// TwinCAT 3 PLC project TcLogger
// Title: TcLogger
// Company: TcLogger
// ProjectVersion: 0.2.0
// ProgramVersion: 3.1.4022.7
// libraries:
//   Tc2_Standard, * (Beckhoff Automation GmbH)
//   Tc2_System, * (Beckhoff Automation GmbH)
//   Tc2_Utilities, * (Beckhoff Automation GmbH)
//   Tc3_Module, * (Beckhoff Automation GmbH)
//   TcExt, * (TcExt)
//   TcUnit, * (www.tcunit.org)
// project tree:
//   Event/ Event.TcPOU (not stored), EventLevel.TcDUT, EventMessage.TcDUT (not stored), EventRunner.TcPOU
//   GVL/ GVL.TcGVL, Properties.TcGVL
//   Logger/ ADSLogger.TcPOU, EventLogger.TcIO, FileLogger.TcPOU, MemoryLogger.TcPOU, run.TcPOU
//   / PlcTask.TcTTO
//   Tests/Event/ EventTestsystem.TcDUT (not stored), MultipleEventTestsystem.TcDUT, TestEvent.TcPOU
//   Tests/Logger/ ADSLoggerTestsystem.TcDUT, TestADSLogger.TcPOU, TestFileLogger.TcPOU
//   Tests/ TEST_MAIN.TcPOU
//   Utils/ F_FIFO_WRITE.TcPOU (not stored), remove_field_from_array.TcPOU (not stored)
// real-time tasks:
//   TASK PlcTask: cycle T#10ms, priority 20, ADS port 350

CONFIGURATION TcLogger
    RESOURCE PLC ON TwinCAT3
        TASK PlcTask(INTERVAL := T#10ms, PRIORITY := 20);
        PROGRAM TEST_MAIN WITH PlcTask : TEST_MAIN;
    END_RESOURCE
END_CONFIGURATION

// ---- Event/EventLevel.TcDUT
{attribute 'qualified_only'}
{attribute 'strict'}
TYPE EventLevel :
(
	INFO := 10,
  WARNING :=20,
  ERROR := 30
) BYTE := INFO;
END_TYPE

// ---- Tests/Event/MultipleEventTestsystem.TcDUT
TYPE MultipleEventTestsystem :
STRUCT
  runner: EventRunner;
  event1: Event := (runner:=runner);
  event2: Event := (runner:=runner);
  event3: Event := (runner:=runner);
END_STRUCT
END_TYPE

// ---- Tests/Logger/ADSLoggerTestsystem.TcDUT
TYPE ADSLoggerTestsystem :
STRUCT
  runner: EventRunner;
  event: Event := (runner:=runner);
  logger: ADSLogger := (disable_ads_output := TRUE);
END_STRUCT
END_TYPE

// ---- GVL/GVL.TcGVL
{attribute 'qualified_only'}
VAR_GLOBAL
  runner: EventRunner;
END_VAR

// ---- GVL/Properties.TcGVL
{attribute 'qualified_only'}
VAR_GLOBAL CONSTANT
  NUM_EVENTS: INT := 4;
  NUM_EVENT_HISTORY: INT := 10;
  NUM_CONCURRENT_ALARMS: INT := 10;
  NUM_LOGGER: INT := 5;
END_VAR

// ---- Logger/EventLogger.TcIO
INTERFACE EventLogger

PROPERTY PUBLIC level : EventLevel
GET
END_GET
SET
END_SET
END_PROPERTY

METHOD PUBLIC submit_event_message
VAR_INPUT
  ev: EventMessage;
END_VAR
END_METHOD

END_INTERFACE

// ---- Tests/TEST_MAIN.TcPOU
PROGRAM TEST_MAIN
VAR
  test_event: TestEvent;
  test_ads_logger: TestADSLogger;
  //test_file_logger: TestFileLogger;
END_VAR

TcUnit.RUN();

END_PROGRAM

// ---- Tests/Event/TestEvent.TcPOU
FUNCTION_BLOCK TestEvent EXTENDS TcUnit.FB_TestSuite
VAR_INPUT
END_VAR
VAR_OUTPUT
END_VAR
VAR
END_VAR

event_erstellen();
//file_logger_testen();
after_initialisation_alarm_is_not_raised();
after_raising_an_alarm_the_alarm_is_raised();
clear_alarm();
add_multiple_events();
raise_and_clear_multiple_alarms();

METHOD add_multiple_events
VAR_INST
  sut: MultipleEventTestsystem;
END_VAR
TEST('Add multiple events');

sut.event1.alarm();
sut.event2.warning();
sut.event3.alarm();
AssertTrue(sut.event1.alarm_raised, 'Event 1');
AssertFalse(sut.event2.alarm_raised, 'Event 2');
AssertTrue(sut.event3.alarm_raised, 'Event 3');

TEST_FINISHED();
END_METHOD

METHOD after_initialisation_alarm_is_not_raised
VAR_INPUT
END_VAR
VAR_INST
  sut: EventTestsystem;
END_VAR
TEST('Alarm is not raised after initialisation');

AssertFalse(sut.event.alarm_raised, '');

TEST_FINISHED();
END_METHOD

METHOD after_raising_an_alarm_the_alarm_is_raised
VAR_INPUT
END_VAR
VAR_INST
  sut: EventTestsystem;
END_VAR
TEST('After raising an alarm the alarm is raised');

sut.event.alarm();
AssertTrue(sut.event.alarm_raised, '');

TEST_FINISHED();
END_METHOD

METHOD clear_alarm
VAR_INPUT
END_VAR
VAR_INST
  sut: EventTestsystem;
END_VAR
TEST('Clear alarm');

sut.event.alarm();
sut.event.clear_alarm();
AssertFalse(sut.event.alarm_raised, '');

TEST_FINISHED();
END_METHOD

METHOD event_erstellen
VAR_INPUT
END_VAR
VAR_INST
  sut: EventTestsystem;
END_VAR
TEST('event_erstellen');

sut.event.message := 'Test';
AssertEquals_STRING('Test', sut.event.message, 'Event not properly created');

TEST_FINISHED();
END_METHOD

METHOD file_logger_testen
VAR_INPUT
END_VAR
VAR_INST
  sut: EventTestsystem;
  file_logger: FileLogger;
END_VAR
TEST('file_logger_testen');

file_logger.path := 'c:\';
sut.runner.add_logger(file_logger);
sut.event.message := 'Test';
sut.event.alarm();

//sut.runner.save_logger(execute:=TRUE);

//IF sut.runner.saving_logger_done() THEN
  TEST_FINISHED();
//END_IF
END_METHOD

METHOD raise_and_clear_multiple_alarms
VAR_INST
  sut: MultipleEventTestsystem;
END_VAR
TEST('Raise and clear multiple alarms');

sut.event1.alarm();
sut.event2.alarm();
sut.event3.alarm();
sut.event1.clear_alarm();
sut.event3.clear_alarm();
AssertFalse(sut.event1.alarm_raised, 'Event 1');
AssertTrue(sut.event2.alarm_raised, 'Event 2');
AssertFalse(sut.event3.alarm_raised, 'Event 3');

TEST_FINISHED();
END_METHOD

END_FUNCTION_BLOCK

// ---- Logger/FileLogger.TcPOU
FUNCTION_BLOCK FileLogger IMPLEMENTS EventLogger
VAR_INPUT
END_VAR
VAR_OUTPUT
  error_id: DWORD;
END_VAR
VAR
  _path: STRING(255);
  file: TcExt.FileMemory;
  localtime: FB_LocalSystemTime := (bEnable:=TRUE);
  _done: BOOL;
  _level: EventLevel;
END_VAR

PROPERTY done : BOOL
GET
done := _done;
END_GET
SET // PRIVATE
_done := done;
END_SET
END_PROPERTY

METHOD PRIVATE get_timestaped_path : STRING(255)
VAR
  datetime: STRING(255);
  char_at: INT;
END_VAR
datetime := SYSTEMTIME_TO_STRING(localtime.systemTime);

char_at := FIND(datetime, '.');
IF char_at <> 0 THEN
  datetime := DELETE(datetime, 4, char_at);
END_IF

REPEAT
  char_at := FIND(datetime, ':');
  IF char_at <> 0 THEN
    datetime := REPLACE(datetime, '_', 1, char_at);
  END_IF
UNTIL char_at = 0
END_REPEAT

get_timestaped_path := CONCAT(path, CONCAT('log_', CONCAT(datetime, '.log')));
END_METHOD

PROPERTY PUBLIC level : EventLevel
GET
level := _level;
END_GET
SET
_level := level;
END_SET
END_PROPERTY

PROPERTY path : STRING(255)
GET
path := _path;
END_GET
SET
_path := path;
END_SET
END_PROPERTY

METHOD save
VAR_INPUT
  execute: BOOL;
  data_ptr: PVOID;
  data_size: DWORD;
END_VAR
VAR_INST
  r_execute: R_TRIG;
END_VAR
localtime();
r_execute(CLK:=execute);

IF r_execute.Q THEN
  file.path := get_timestaped_path();
END_IF
file.write(
  start:=execute,
  data_ptr:=data_ptr,
  data_size:=data_size,
  done=>_done,
  error_id=>error_id);
END_METHOD

METHOD submit_event_message
VAR_INPUT
	ev: EventMessage;
END_VAR
END_METHOD

END_FUNCTION_BLOCK

// ---- Tests/Logger/TestADSLogger.TcPOU
FUNCTION_BLOCK TestADSLogger EXTENDS TcUnit.FB_TestSuite
VAR_INPUT
END_VAR
VAR_OUTPUT
END_VAR
VAR
END_VAR

submit_info();
submit_warning();
submit_error();
submit_alarm();

METHOD submit_alarm
VAR_INPUT
END_VAR
VAR_INST
  sut: ADSLoggerTestsystem;
END_VAR
TEST('Submit alarm');

sut.runner.add_logger(sut.logger);
sut.event.message := 'Alarm';
sut.event.alarm();

AssertEquals_DWORD(ADSLOG_MSGTYPE_ERROR, sut.logger.mask, '');
AssertEquals_STRING(' | Error: ', sut.logger.prefix, '');
AssertEquals_STRING(' | Error: Alarm', sut.logger.formatted_output, '');

TEST_FINISHED();
END_METHOD

METHOD submit_error
VAR_INPUT
END_VAR
VAR_INST
  sut: ADSLoggerTestsystem;
END_VAR
TEST('Submit error');

sut.runner.add_logger(sut.logger);
sut.event.message := 'Error';
sut.event.error();

AssertEquals_DWORD(ADSLOG_MSGTYPE_ERROR, sut.logger.mask, '');
AssertEquals_STRING(' | Error: ', sut.logger.prefix, '');
AssertEquals_STRING(' | Error: Error', sut.logger.formatted_output, '');

TEST_FINISHED();
END_METHOD

METHOD submit_info
VAR_INPUT
END_VAR
VAR_INST
  sut: ADSLoggerTestsystem;
END_VAR
TEST('Submit info');

sut.runner.add_logger(sut.logger);
sut.event.message := 'Info';
sut.event.info();

AssertEquals_DWORD(ADSLOG_MSGTYPE_HINT, sut.logger.mask, '');
AssertEquals_STRING(' | Info: ', sut.logger.prefix, '');
AssertEquals_STRING(' | Info: Info', sut.logger.formatted_output, '');

TEST_FINISHED();
END_METHOD

METHOD submit_warning
VAR_INPUT
END_VAR
VAR_INST
  sut: ADSLoggerTestsystem;
END_VAR
TEST('Submit warning');

sut.runner.add_logger(sut.logger);
sut.event.message := 'Warning';
sut.event.warning();

AssertEquals_DWORD(ADSLOG_MSGTYPE_WARN, sut.logger.mask, '');
AssertEquals_STRING(' | Warning: ', sut.logger.prefix, '');
AssertEquals_STRING(' | Warning: Warning', sut.logger.formatted_output, '');

TEST_FINISHED();
END_METHOD

END_FUNCTION_BLOCK

// ---- Logger/run.TcPOU
PROGRAM run
VAR
END_VAR

GVL.runner.run(disable_ads_output:=TRUE);

END_PROGRAM

// ---- Event/EventRunner.TcPOU
FUNCTION_BLOCK EventRunner
VAR_INPUT
END_VAR
VAR_OUTPUT
END_VAR
VAR
  event_id_counter: INT;
  localtime: FB_LocalSystemTime := (bEnable:=TRUE);
  actSystemTime: TIMESTRUCT;
  event_logger: ARRAY [1..Properties.NUM_LOGGER] OF EventLogger;
  active_alarms: ARRAY[1..Properties.NUM_CONCURRENT_ALARMS] OF EventMessage;
  logger_counter: INT;
END_VAR

(* 
der runner wird am ende des sps programms ausgefuehrt
- als input kommt das signal zum sichern der daten (bei der cx81xx bspw. das signal der usv). diese werden binaer gesichtert, koennen jedoch zusaetzlich als csv gesichert werden
- ansonsten kuemmert sich der runner nur um die erstellung eines arrays zur darstellung in einer hmi mit den aktuell aktiven events
- im programm werden pro meldung event-instanzen erstellt. diese registrieren sich selbst. die richtige id wird der pfad zur instanzvariable sein
- im runner wird zudem das datum immer aktualisiert
*)

PROPERTY PRIVATE act_time : TIMESTRUCT
GET
IF time_valid THEN
  act_time := localtime.systemTime;
END_IF
END_GET
END_PROPERTY

METHOD PUBLIC add_logger
VAR_INPUT
  logger: EventLogger;
END_VAR
IF logger_counter < Properties.NUM_LOGGER AND ADR(logger) <> 0 THEN
  inc_logger_counter();
  event_logger[logger_counter] := logger;
END_IF
END_METHOD

METHOD INTERNAL alarm_raised : BOOL
VAR_INPUT
  id: INT;
END_VAR
VAR
  i: INT;
END_VAR
alarm_raised := get_alarm_index(id:=id) > 0;
END_METHOD

METHOD INTERNAL clear_alarm
VAR_INPUT
  id: INT;
END_VAR
VAR
  index: INT;
  filldata: EventMessage;
END_VAR
IF alarm_raised(id:=id) THEN
  index := get_alarm_index(id:=id);
  active_alarms[index].timestamp_cleared := act_time;
  active_alarms[index].cleared := TRUE;
  
  submit_event_message_to_logger(active_alarms[index]);
  
  remove_field_from_array(
    index_to_remove:=index,
    size_filldata:=SIZEOF(filldata),
    adr_filldata:=ADR(filldata),
    size_memory_buffer:=SIZEOF(active_alarms),
    adr_memory_buffer:=ADR(active_alarms));
END_IF
END_METHOD

METHOD PRIVATE create_event_message : EventMessage
VAR_INPUT
  id: INT;
  message: STRING(255);
  level: EventLevel;
  cleared: BOOL;
END_VAR
VAR
  ev: EventMessage;
  undefined_time: TIMESTRUCT;
END_VAR
ev.id := id;
ev.message := message;
ev.level := level;
ev.cleared := cleared;
ev.timestamp_raised := act_time;
IF cleared THEN
  ev.timestamp_cleared := act_time;
ELSE
  ev.timestamp_cleared := undefined_time;
END_IF

create_event_message := ev;
END_METHOD

METHOD INTERNAL generate_event_id : INT
VAR_INPUT
END_VAR
inc_event_id_counter();
generate_event_id := event_id_counter;
END_METHOD

METHOD PRIVATE get_alarm_index : INT
VAR_INPUT
  id: INT;
END_VAR
VAR
  i: INT;
END_VAR
get_alarm_index := 0;
FOR i:=1 TO Properties.NUM_EVENT_HISTORY DO
  IF active_alarms[i].id = id AND NOT active_alarms[i].cleared THEN
    get_alarm_index := i;
    EXIT;
	END_IF
END_FOR
END_METHOD

METHOD PRIVATE inc_event_id_counter
VAR_INPUT
END_VAR
event_id_counter := LIMIT(1, event_id_counter + 1, Properties.NUM_EVENTS);
END_METHOD

METHOD PRIVATE inc_logger_counter
VAR_INPUT
END_VAR
logger_counter := LIMIT(1, logger_counter + 1, Properties.NUM_LOGGER);
END_METHOD

METHOD INTERNAL raise_alarm
VAR_INPUT
  id: INT;
  message: STRING(255);
  level: EventLevel;
END_VAR
VAR
  undefined_time: TIMESTRUCT;
END_VAR
IF NOT alarm_raised(id:=id) THEN
  submit_event_message(
    id:=id,
    message:=message,
    level:=level,
    cleared:=FALSE);
END_IF
END_METHOD

METHOD run
VAR_INPUT
END_VAR
VAR
  read_done: BOOL;
  error_id: UDINT;
END_VAR
localtime();
END_METHOD

METHOD PRIVATE submit_event_message
VAR_INPUT
  id: INT;
  message: STRING(255);
  level: EventLevel;
  cleared: BOOL;
END_VAR
VAR
  ev: EventMessage;
END_VAR
ev := create_event_message(id, message, level, cleared);

F_FIFO_WRITE(SIZEOF(ev), ADR(ev), SIZEOF(active_alarms), ADR(active_alarms));

submit_event_message_to_logger(ev);
END_METHOD

METHOD PRIVATE submit_event_message_to_logger
VAR_INPUT
  ev: EventMessage;
END_VAR
VAR
  i: INT;
END_VAR
FOR i:=1 TO Properties.NUM_LOGGER DO
  IF event_logger[i] <> 0 THEN
    event_logger[i].submit_event_message(ev);
	END_IF
END_FOR
END_METHOD

METHOD INTERNAL submit_message
VAR_INPUT
  id: INT;
  message: STRING(255);
  level: EventLevel;
END_VAR
submit_event_message(
  id:=id,
  message:=message,
  level:=level,
  cleared:=TRUE);
END_METHOD

PROPERTY PUBLIC time_valid : BOOL
GET // PRIVATE
time_valid := localtime.bValid;
END_GET
END_PROPERTY

METHOD PRIVATE timestruct_equal : BOOL
VAR_INPUT
  timestruct_1: TIMESTRUCT;
  timestruct_2: TIMESTRUCT;
END_VAR
timestruct_equal := timestruct_1.wDay = timestruct_2.wDay;
timestruct_equal := timestruct_equal AND timestruct_1.wDayOfWeek = timestruct_2.wDayOfWeek;
timestruct_equal := timestruct_equal AND timestruct_1.wHour = timestruct_2.wHour;
timestruct_equal := timestruct_equal AND timestruct_1.wMilliseconds = timestruct_2.wMilliseconds;
timestruct_equal := timestruct_equal AND timestruct_1.wMinute = timestruct_2.wMinute;
END_METHOD

END_FUNCTION_BLOCK

// ---- Logger/ADSLogger.TcPOU
FUNCTION_BLOCK ADSLogger IMPLEMENTS EventLogger
VAR_INPUT
END_VAR
VAR_OUTPUT
END_VAR
VAR
  _level: EventLevel;
  _disable_ads_output: BOOL;
  _mask: DWORD;
  _prefix: STRING(15);
  _formatted_output: STRING(255);
END_VAR

METHOD PRIVATE ads_log
VAR_INPUT
  ev: EventMessage;
END_VAR
VAR
END_VAR
mask := create_mask(ev.level);
prefix := create_prefix(ev.level);

formatted_output := CONCAT(prefix, ev.message);

IF NOT disable_ads_output THEN
  ADSLOGSTR(mask, formatted_output, '');
END_IF
END_METHOD

METHOD PRIVATE create_mask : DWORD
VAR_INPUT
  level: EventLevel;
END_VAR
CASE level OF
EventLevel.INFO:
  create_mask := ADSLOG_MSGTYPE_HINT;
EventLevel.WARNING:
  create_mask := ADSLOG_MSGTYPE_WARN;
EventLevel.ERROR:
  create_mask := ADSLOG_MSGTYPE_ERROR;
ELSE
  create_mask := ADSLOG_MSGTYPE_HINT;
END_CASE
END_METHOD

METHOD PRIVATE create_prefix : STRING(15)
VAR_INPUT
  level: EventLevel;
END_VAR
CASE level OF
EventLevel.INFO:
  create_prefix := ' | Info: ';
EventLevel.WARNING:
  create_prefix := ' | Warning: ';
EventLevel.ERROR:
  create_prefix := ' | Error: ';
ELSE
  create_prefix := ' | Undefined: ';
END_CASE
END_METHOD

PROPERTY INTERNAL disable_ads_output : BOOL
GET
disable_ads_output := _disable_ads_output;
END_GET
SET
_disable_ads_output := disable_ads_output;
END_SET
END_PROPERTY

PROPERTY INTERNAL formatted_output : STRING(255)
GET
formatted_output := _formatted_output;
END_GET
SET // PRIVATE
_formatted_output := formatted_output;
END_SET
END_PROPERTY

PROPERTY PUBLIC level : EventLevel
GET
level := _level;
END_GET
SET
_level := level;
END_SET
END_PROPERTY

PROPERTY INTERNAL mask : DWORD
GET
mask := _mask;
END_GET
SET // PRIVATE
_mask := mask;
END_SET
END_PROPERTY

PROPERTY INTERNAL prefix : STRING(15)
GET
prefix := _prefix;
END_GET
SET // PRIVATE
_prefix := prefix;
END_SET
END_PROPERTY

METHOD PUBLIC submit_event_message
VAR_INPUT
	ev: EventMessage;
END_VAR
IF ev.level >= level THEN
  ads_log(ev);
END_IF
END_METHOD

END_FUNCTION_BLOCK

// ---- Logger/MemoryLogger.TcPOU
FUNCTION_BLOCK MemoryLogger IMPLEMENTS EventLogger
VAR_INPUT
END_VAR
VAR_OUTPUT
END_VAR
VAR
  event_history: ARRAY[1..Properties.NUM_EVENT_HISTORY] OF EventMessage;
END_VAR

METHOD submit_event_message
VAR_INPUT
	ev: EventMessage;
END_VAR
F_FIFO_WRITE(SIZEOF(ev), ADR(ev), SIZEOF(event_history), ADR(event_history));
END_METHOD

END_FUNCTION_BLOCK

// ---- Tests/Logger/TestFileLogger.TcPOU
FUNCTION_BLOCK TestFileLogger EXTENDS TcUnit.FB_TestSuite
VAR_INPUT
END_VAR
VAR_OUTPUT
END_VAR
VAR
END_VAR

END_FUNCTION_BLOCK
